FUNCTION_BLOCK AUDI_AUI_DEMUX_3_UNGATED (* Wie AUDI_AUI_DEMUX_3, aber OHNE Aenderungserkennung - reicht JEDES neu berechnete Ergebnis bedingungslos weiter (fuer Verbraucher, die eine periodische Kadenz unabhaengig von Wertaenderung brauchen, z.B. Ableitungs-/Frequenzberechnungen). (AUDI demultiplexor (generic FB)) *)
  (* Standard: 61499-2; Description: Copyright (c) 2026 Meisterschulen am Ostbahnhof This program and the accompanying materials are made available under the terms of the Eclipse Public License 2.0 which is available at https://www.eclipse.org/legal/epl-2.0/ SPDX-License-Identifier: EPL-2.0 *)
  (* Version 1.0, 2026-08-31, Franz Höpfinger, HR Agrartechnik GmbH *)
  PACKAGE adapter::selection::unidirectional;
  {SET_ATTRIBUTE(eclipse4diac::core::GenericClassName, 'GEN_AUDI_AUI_DEMUX')}
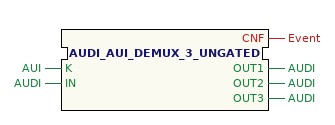
  EVENT_OUTPUT
    CNF; (* Confirmation of Set Index K *)
  END_EVENT
  SOCKETS
    K : adapter::types::unidirectional::AUI; (* index *)
    IN : adapter::types::unidirectional::AUDI; (* Input Value to demultiplex *)
  END_SOCKETS
  PLUGS
    OUT1 : adapter::types::unidirectional::AUDI; (* Output value 1 (selected when K = 0) *)
    OUT2 : adapter::types::unidirectional::AUDI; (* Output value 2 (selected when K = 1) *)
    OUT3 : adapter::types::unidirectional::AUDI; (* Output value 3 (selected when K = 2) *)
  END_PLUGS
END_FUNCTION_BLOCK
